# EPICS autosave request: psdPortDriverApp/Db/psdPortDriver_settings.req
# This file is used by autosave to determine what PVs to save

$(P)$(R)Connect
$(P)$(R)AcquireTime
$(P)$(R)NBins
$(P)$(R)Mode
$(P)$(R)SoftLLD
$(P)$(R)SoftHLD
$(P)$(R)HardLLD
